PROGRAM Mode_Call
VAR
	FB_ModeMang: FB_ModeCall;
	tAlwaysOff:bool;
	TON_0: TON;
	FB_Roller_Door_1: FB_Roller_Door;
	FB_Roller_Door_2: FB_Roller_Door;
	FB_TurnTable_0_180_0: FB_TurnTable_0_180;
END_VAR

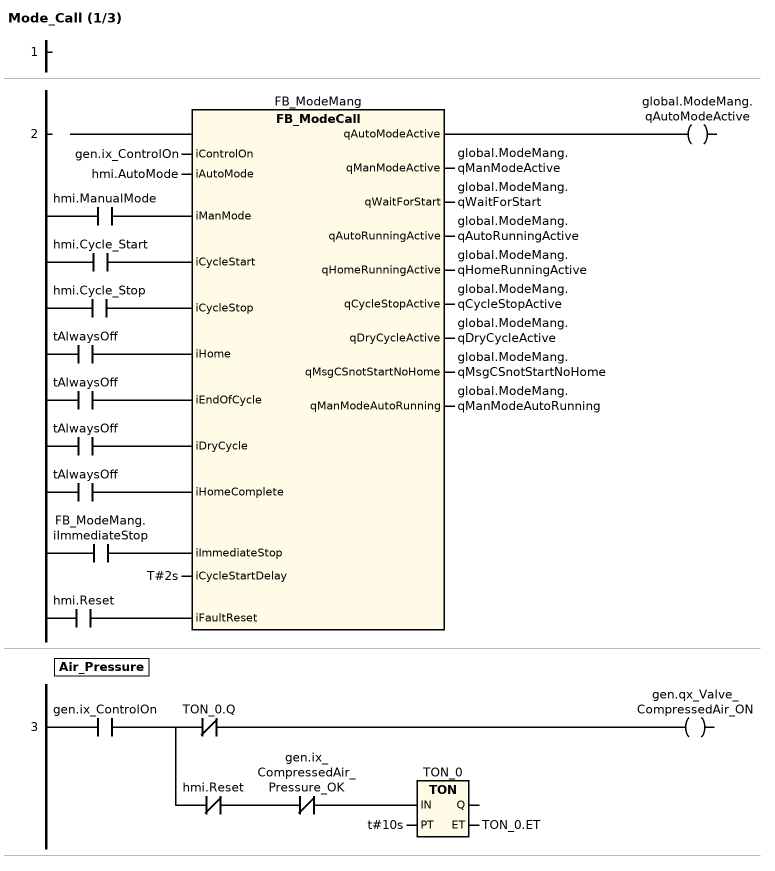
// NETWORK 1

// NETWORK 2
FB_ModeMang(
    iControlOn := gen.ix_ControlOn,
    iAutoMode := hmi.AutoMode,
    iManMode := hmi.ManualMode,
    iCycleStart := hmi.Cycle_Start,
    iCycleStop := hmi.Cycle_Stop,
    iHome := tAlwaysOff,
    iEndOfCycle := tAlwaysOff,
    iDryCycle := tAlwaysOff,
    iHomeComplete := tAlwaysOff,
    iImmediateStop := FB_ModeMang.iImmediateStop,
    iCycleStartDelay := T#2s,
    iFaultReset := hmi.Reset,
    qManModeActive => global.ModeMang.qManModeActive,
    qWaitForStart => global.ModeMang.qWaitForStart,
    qAutoRunningActive => global.ModeMang.qAutoRunningActive,
    qHomeRunningActive => global.ModeMang.qHomeRunningActive,
    qCycleStopActive => global.ModeMang.qCycleStopActive,
    qDryCycleActive => global.ModeMang.qDryCycleActive,
    qMsgCSnotStartNoHome => global.ModeMang.qMsgCSnotStartNoHome,
    qManModeAutoRunning => global.ModeMang.qManModeAutoRunning); // FB_ModeCall
global.ModeMang.qAutoModeActive := FB_ModeMang.qAutoModeActive;

// NETWORK 3
Air_Pressure:
gen.qx_Valve_CompressedAir_ON := gen.ix_ControlOn AND NOT TON_0.Q;
TON_0(
    IN := gen.ix_ControlOn AND NOT hmi.Reset AND NOT gen.ix_CompressedAir_Pressure_OK,
    PT := t#10s,
    ET => TON_0.ET); // TON

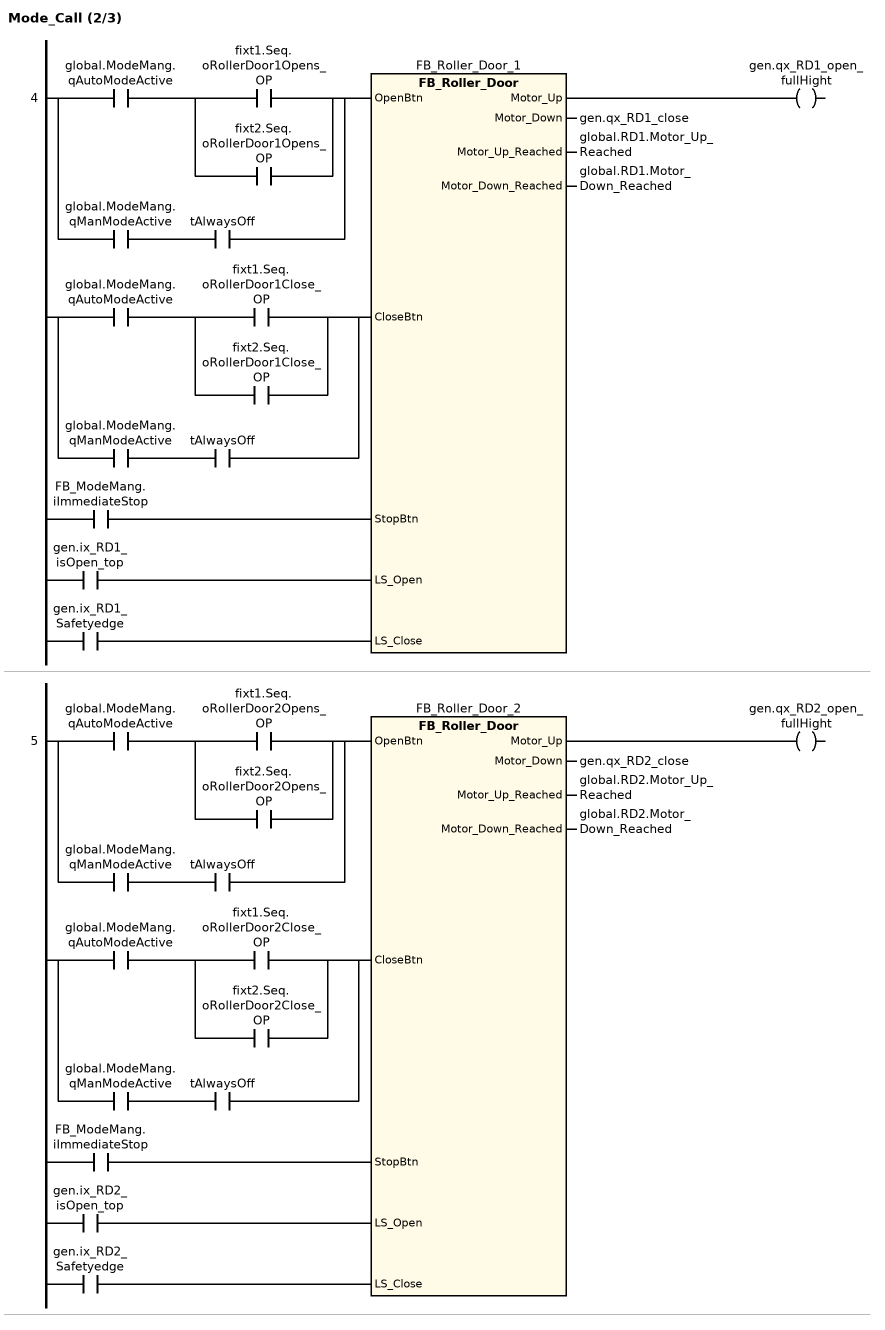
// NETWORK 4
FB_Roller_Door_1(
    OpenBtn := global.ModeMang.qAutoModeActive AND (fixt1.Seq.oRollerDoor1Opens_OP OR fixt2.Seq.oRollerDoor1Opens_OP) OR global.ModeMang.qManModeActive AND tAlwaysOff,
    CloseBtn := global.ModeMang.qAutoModeActive AND (fixt1.Seq.oRollerDoor1Close_OP OR fixt2.Seq.oRollerDoor1Close_OP) OR global.ModeMang.qManModeActive AND tAlwaysOff,
    StopBtn := FB_ModeMang.iImmediateStop,
    LS_Open := gen.ix_RD1_isOpen_top,
    LS_Close := gen.ix_RD1_Safetyedge,
    Motor_Down => gen.qx_RD1_close,
    Motor_Up_Reached => global.RD1.Motor_Up_Reached,
    Motor_Down_Reached => global.RD1.Motor_Down_Reached); // FB_Roller_Door
gen.qx_RD1_open_fullHight := FB_Roller_Door_1.Motor_Up;

// NETWORK 5
FB_Roller_Door_2(
    OpenBtn := global.ModeMang.qAutoModeActive AND (fixt1.Seq.oRollerDoor2Opens_OP OR fixt2.Seq.oRollerDoor2Opens_OP) OR global.ModeMang.qManModeActive AND tAlwaysOff,
    CloseBtn := global.ModeMang.qAutoModeActive AND (fixt1.Seq.oRollerDoor2Close_OP OR fixt2.Seq.oRollerDoor2Close_OP) OR global.ModeMang.qManModeActive AND tAlwaysOff,
    StopBtn := FB_ModeMang.iImmediateStop,
    LS_Open := gen.ix_RD2_isOpen_top,
    LS_Close := gen.ix_RD2_Safetyedge,
    Motor_Down => gen.qx_RD2_close,
    Motor_Up_Reached => global.RD2.Motor_Up_Reached,
    Motor_Down_Reached => global.RD2.Motor_Down_Reached); // FB_Roller_Door
gen.qx_RD2_open_fullHight := FB_Roller_Door_2.Motor_Up;

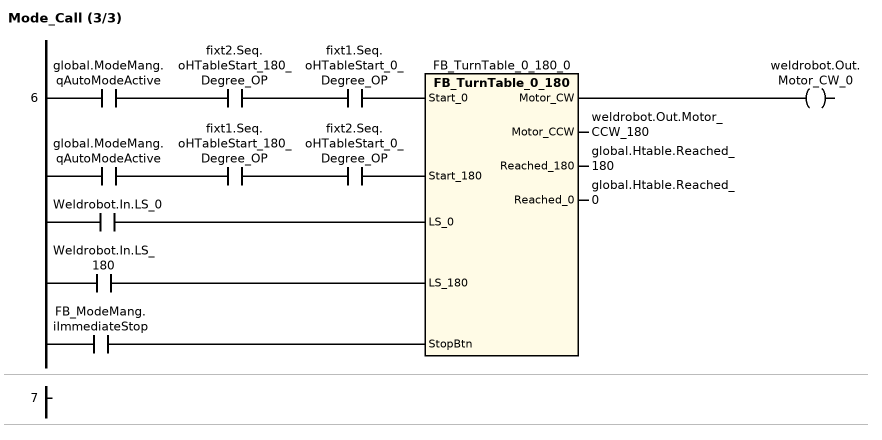
// NETWORK 6
FB_TurnTable_0_180_0(
    Start_0 := global.ModeMang.qAutoModeActive AND fixt2.Seq.oHTableStart_180_Degree_OP AND fixt1.Seq.oHTableStart_0_Degree_OP,
    Start_180 := global.ModeMang.qAutoModeActive AND fixt1.Seq.oHTableStart_180_Degree_OP AND fixt2.Seq.oHTableStart_0_Degree_OP,
    LS_0 := Weldrobot.In.LS_0,
    LS_180 := Weldrobot.In.LS_180,
    StopBtn := FB_ModeMang.iImmediateStop,
    Motor_CCW => weldrobot.Out.Motor_CCW_180,
    Reached_180 => global.Htable.Reached_180,
    Reached_0 => global.Htable.Reached_0); // FB_TurnTable_0_180
weldrobot.Out.Motor_CW_0 := FB_TurnTable_0_180_0.Motor_CW;

// NETWORK 7

END_PROGRAM

(* stored: Version 1.1.0.1, ProductVersion 3.1.4024.16
   POU Mode_Call: Id {4809c63a-e255-4adb-a8ec-f5d9117b0ba1}, SpecialFunc None *)
